Staubli VAL3: DAEMON2.PGX

public program daemon2()
  local jointRx l_jCurr
  local num l_i
  local bool l_bError
  local string l_sMsg
  local num l_nError
  local bool l_bDrivesOK
begin

  // Verification du bit de vie bus can
  call chkLifeBit()

  // Gestion watchDog pour variateurs
  //call updateWatchDog()
  //
  // Recupere etat des variateurs
  l_bDrivesOK=true
  for l_i=0 to nNUMOFAXES-1
    bDrvFault[l_i]=(diFault[l_i]==true) or bAnd(aioGet(aiStatusRemote[l_i])/32,255)!=0
    call chkDrvState(l_i)
    l_bDrivesOK=l_bDrivesOK and nDrvState[l_i]==cst:nOperatEnabled
    bDrivesOpEnable=l_bDrivesOK
  endFor

  if isPowered() and l_bDrivesOK
    // Get system position
    $XgetDrvCmdPos(nDrvPos)
    l_sMsg=""
    //$XgetJntCmdPos(l_nJntPos)
    for l_i=0 to nNUMOFAXES-1
      // Send it to the external axis
      aioSet(aoPosCmd[l_i],nDrvPos[l_i]*nScaleFact)
      //l_sMsg="0: "+toString(".3",l_nJntPos[0])+"   1: "+toString(".3",l_nJntPos[1])
      l_sMsg=l_sMsg+toString("",l_i)+": "+toString(".3",nDrvPos[l_i])+"   "
    endFor
    //? l_sMsg
  else
    for l_i=0 to nNUMOFAXES-1
      doEnableOp[l_i]=false
      doSwitchOn[l_i]=false
      // Get external axis position
      nDrvPos[l_i]=aioGet(aiPosFbk[l_i])/nScaleFact
    endFor
    // Update it in the system
    $XsetDrvFbkPos(nDrvPos)
  endIf



end
